// TIA Portal V20 export
DATA_BLOCK "CallEquipment_DB"   // DB158
{ DB_Accessible_From_OPC_UA := 'FALSE' }
// stored: AssignedProDiagFB Unit1.Em1.ProDiag, DBAccessibleFromOPCUA false, DBAccessibleFromWebserver false, InstanceOfName Unit1.Em1.CallEquipment, InstanceOfType FB, Namespace Unit1.Em1
"Unit1.Em1.CallEquipment"
   // VAR_INPUT
   //    ZoneOperationEnable { ExternalWritable := 'False'} : "LWONIK_typeSafetyZoneManualOperation";
   // END_VAR
   // VAR_IN_OUT
   //    unitStatus : "LAF_typeUnitStatus";
   //    emFeedback : "LUC_typeEmFeedback";
   //    unitAlarmDB : "LAF_typeAlarms";
   // END_VAR
   // VAR
   //    InstStacker2NgBoxSequence { ExternalWritable := 'False'} : "Unit1.Em1.Sequence_1_Stacker2NgBox";
   //    instStacker2NgBoxHomeJob1 { ExternalWritable := 'False'} : "LAF_SelectJob";
   //    instStacker2NgBoxLoadJob2 { ExternalWritable := 'False'} : "LAF_SelectJob";
   //    instStacker2NgBoxUnloadJob3 { ExternalWritable := 'False'} : "LAF_SelectJob";
   //    instCmStacker2NgBoxDetect { ExternalWritable := 'False'} : "LBC_DigitalSignalCn";
   //    instCmStacker2NgBoxFullDetect { ExternalWritable := 'False'} : "LBC_DigitalSignalCn";
   //    instStacker2NgBoxLoadingUpDown { ExternalWritable := 'False'} : "LBC_TwoWayActuatorCn";
   //    instStacker2NgBoxUnitMoverBwdFwd { ExternalWritable := 'False'} : "LBC_TwoWayActuatorCn";
   //    instStacker2NgBoxClampLeftOpenClose { ExternalWritable := 'False'} : "LBC_TwoWayActuatorCn";
   //    instStacker2NgBoxClampRightOpenClose { ExternalWritable := 'False'} : "LBC_TwoWayActuatorCn";
   //    instStacker2NgBoxClampMoverOpenClose { ExternalWritable := 'False'} : "LBC_TwoWayActuatorCn";
   //    instStacker2NgBoxLiftDownUp { ExternalWritable := 'False'} : "LBC_TwoWayActuatorCn";
   //    instStacker2NgBoxLockDownUp { ExternalWritable := 'False'} : "LBC_TwoWayActuatorCn";
   //    instManageAlarms { ExternalWritable := 'False'} : "LAF_ManageAlarms";
   //    instEventsPFE { ExternalWritable := 'False'} : "Unit1.Em1.EventsPFE";
   //    statUnitStatus { ExternalWritable := 'False'} : "LAF_typeUnitStatus";
   //    statTonTime { ExternalWritable := 'False'} : Array[0..999] of TON_TIME;
   //    statTofTime { ExternalWritable := 'False'} : Array[0..99] of TOF_TIME;
   //    statPulse { ExternalWritable := 'False'} : Array[0..999] of Bool;
   //    statEnableManualCmds { ExternalWritable := 'False'} : Bool;
   //    "*** Interlock TwoWay ***" { S7_SetPoint := 'True'} : "LER_Axis_Homing";
   //    instCmStacker2NgBoxLoadingUpDownInterlock { S7_SetPoint := 'True'} : Array[0..2] of "LER_Actuator";
   //    instCmStacker2NgBoxUnitMoverBwdFwdInterlock { S7_SetPoint := 'True'} : Array[0..2] of "LER_Actuator";
   //    instCmStacker2NgBoxClampLeftOpenCloseInterlock { S7_SetPoint := 'True'} : Array[0..2] of "LER_Actuator";
   //    instCmStacker2NgBoxClampRightOpenCloseInterlock { S7_SetPoint := 'True'} : Array[0..2] of "LER_Actuator";
   //    instCmStacker2NgBoxClampMoverOpenCloseInterlock { S7_SetPoint := 'True'} : Array[0..2] of "LER_Actuator";
   //    instCmStacker2NgBoxLiftDownUpInterlock { S7_SetPoint := 'True'} : Array[0..2] of "LER_Actuator";
   //    instCmStacker2NgBoxLockDownUpInterlock { S7_SetPoint := 'True'} : Array[0..2] of "LER_Actuator";
   //    instCmStacker2NgBoxLoadingUpDown_IntPos : Array[0..2] of Struct
   //       "Int" : Array[1..10] of Bool;
   //    END_STRUCT;
   //    instCmStacker2NgBoxUnitMoverBwdFwd_IntPos : Array[0..2] of Struct
   //       "Int" : Array[1..10] of Bool;
   //    END_STRUCT;
   //    instCmStacker2NgBoxClampLeftOpenClose_IntPos : Array[0..2] of Struct
   //       "Int" : Array[1..10] of Bool;
   //    END_STRUCT;
   //    instCmStacker2NgBoxClampRightOpenClose_IntPos : Array[0..2] of Struct
   //       "Int" : Array[1..10] of Bool;
   //    END_STRUCT;
   //    instCmStacker2NgBoxClampMoverOpenClose_IntPos : Array[0..2] of Struct
   //       "Int" : Array[1..10] of Bool;
   //    END_STRUCT;
   //    instCmStacker2NgBoxLiftDownUp_IntPos : Array[0..2] of Struct
   //       "Int" : Array[1..10] of Bool;
   //    END_STRUCT;
   //    instCmStacker2NgBoxLockDownUp_IntPos : Array[0..2] of Struct
   //       "Int" : Array[1..10] of Bool;
   //    END_STRUCT;
   //    citi_Ptrig : Array[0..20] of Bool;
   //    citiTon : Array[0..20] of TON_TIME;
   //    citi : Time;
   //    citiTest : Array[0..20] of Bool;
   // END_VAR
BEGIN
END_DATA_BLOCK
